TYPE ST_ProBoxSafetyAK :
STRUCT
	Inputs	AT %I* : ST_ProBoxSafetyInputsAK;
	Outputs AT %Q* : ST_ProBoxSafetyOutputsAK;
END_STRUCT
END_TYPE

(* stored: Version 1.1.0.1, ProductVersion 3.1.4024.4
   DUT ST_ProBoxSafetyAK: Id {ccbea1f2-b80d-4050-81a1-94eb6c9c4088} *)
